PROGRAM P_Queue
VAR
END_VAR

P_Dynamic_Array_Queue();
P_Linked_List_Queue();

END_PROGRAM

(* stored: Version 1.1.0.1, ProductVersion 3.1.4024.4
   POU P_Queue: Id {56cfd7ab-2ed9-4783-a5e7-8ebb28be2ed0}, SpecialFunc None *)
